(* PLC project TEST.project, CODESYS CODESYS V3.5 SP3 Patch 7 *)
(* stored: creationDateTime 2013-12-18T18:39:57.7805164, modificationDateTime 2013-12-11T14:45:29.6582473 *)

FUNCTION_BLOCK Bearbeitungswerkzeug
  VAR
    MOtor : INT;
    Links : INT;
    Rechts : INT;
    Ende : INT;
    Bearbeitung : INT;
  END_VAR

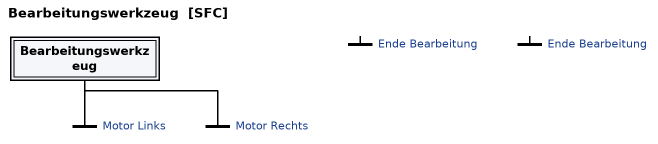
INITIAL_STEP Bearbeitungswerkzeug:
END_STEP
TRANSITION FROM Bearbeitungswerkzeug TO WZ LINKS
  := Motor Links;
END_TRANSITION
TRANSITION FROM Bearbeitungswerkzeug TO WZ RECHTS
  := Motor Rechts;
END_TRANSITION
STEP WZ LINKS:
END_STEP
TRANSITION FROM WZ LINKS TO Init
  := Ende Bearbeitung;
END_TRANSITION
STEP WZ RECHTS:
END_STEP
TRANSITION FROM WZ RECHTS TO Init
  := Ende Bearbeitung;
END_TRANSITION
END_FUNCTION_BLOCK
